Universal Robots PolyScope program: gravityFeederT.urp

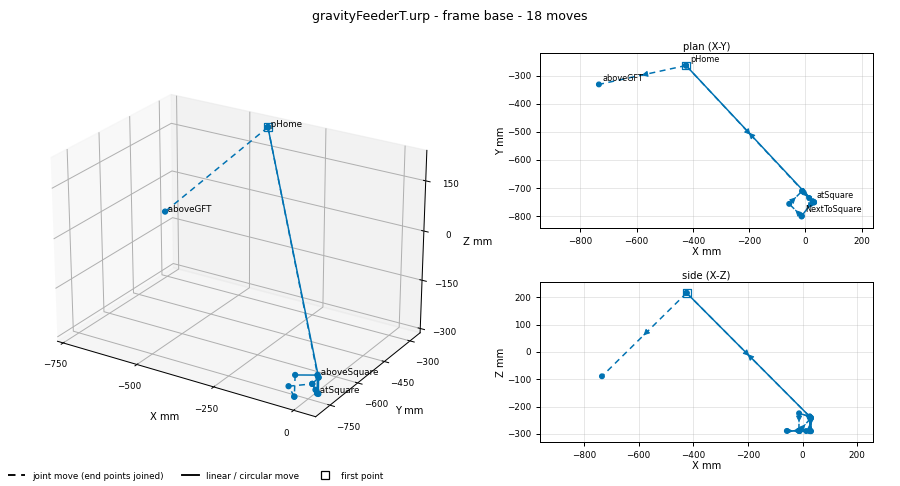
[picture p0: tool path of gravityFeederT.urp in frame base, 18 of 22 moves have a stored position in this frame; points joined in program order, loops and branches not executed]
Program gravityFeederT (installation=admin directory=/programs/THU_530PM createdIn=3.8.0.61336 lastSavedIn=3.15.8.106339 robotSerialNumber=2015350925)
Calibrated DH parameters: a=[0, -0.425, -0.39225, 0, 0, 0]; d=[0.089159, 0, 0, 0.10915, 0.09465, 0.0823]; alpha=[1.570796, 0, 0, 1.570796, -1.570796, 0]; deltaTheta=[0, 0, 0, 0, 0, 0]
Robot Program (runOnlyOnce=true)
  Set DigitalOutput pin=digital_out[0]; digitalValue=0
  Call _adminLinearIndex3
  MoveJ speed 180 deg/s, acceleration 100 deg/s^2 (useActiveTCP=true)
    Waypoint pHome: TCP in base x=-424.182 y=-264.292 z=215.908 mm, rx=-1.1973 ry=-2.8916 rz=-0.0083 rad; joints [224.997, -90.003, -90.003, -90.012, 89.253, -0.016] deg; flange x=-422.241 y=-266.331 z=431.79 mm, rx=-1.1973 ry=-2.8916 rz=-0.0083 rad
    Waypoint aboveGFT: TCP in base x=-733.795 y=-331.415 z=-88.949 mm, rx=-1.1406 ry=-2.7542 rz=0.4281 rad; joints [210.705, -134.689, -80.34, -37.4, 93.732, -13.725] deg; flange x=-685.048 y=-286.122 z=116.441 mm, rx=-1.1406 ry=-2.7542 rz=0.4281 rad
  MoveL speed 250 mm/s, acceleration 1200 mm/s^2 (useActiveTCP=true) feature=Base
    Waypoint atGFRel (Relative): relativeFromPosition TCP in base x=-734.776 y=-331.124 z=-89.043 mm, rx=-1.1456 ry=-2.7528 rz=0.4318 rad; joints [210.705, -134.689, -80.338, -37.4, 93.734, -13.726] deg; TCP in base x=-741.914 y=-341.01 z=-133.241 mm, rx=-1.1403 ry=-2.7544 rz=0.4285 rad; joints [211.023, -139.56, -78.724, -34.121, 93.656, -13.432] deg; flange x=-693.193 y=-295.644 z=72.139 mm, rx=-1.1403 ry=-2.7544 rz=0.4285 rad
    Set DigitalOutput pin=digital_out[0]; digitalValue=1
    Wait Sleep waitTime=1
    Waypoint moveUpRel (Relative): relativeFromPosition TCP in base x=-745.208 y=-342.748 z=-132.176 mm, rx=-1.1455 ry=-2.7527 rz=0.4317 rad; joints [211.078, -139.779, -78.056, -34.566, 93.626, -13.379] deg; TCP in base x=-747.389 y=-346.382 z=-130.447 mm, rx=-1.1404 ry=-2.7544 rz=0.4284 rad; joints [211.165, -140.11, -77.082, -35.205, 93.609, -13.293] deg; flange x=-698.665 y=-301.034 z=74.937 mm, rx=-1.1404 ry=-2.7544 rz=0.4284 rad
    Waypoint aboveGFRel (Relative): relativeFromPosition TCP in base x=-748.436 y=-346.052 z=-130.498 mm, rx=-1.1455 ry=-2.7528 rz=0.432 rad; joints [211.166, -140.109, -77.077, -35.205, 93.607, -13.294] deg; TCP in base x=-735.018 y=-332.975 z=-79.921 mm, rx=-1.1405 ry=-2.7541 rz=0.4282 rad; joints [210.763, -134.184, -79.714, -38.519, 93.714, -13.672] deg; flange x=-686.249 y=-287.668 z=125.46 mm, rx=-1.1405 ry=-2.7541 rz=0.4282 rad
  MoveJ speed 60 deg/s, acceleration 80 deg/s^2 (useActiveTCP=true)
    Waypoint pHome: TCP in base x=-424.182 y=-264.292 z=215.908 mm, rx=-1.1973 ry=-2.8916 rz=-0.0083 rad; joints [224.997, -90.003, -90.003, -90.012, 89.253, -0.016] deg; flange x=-422.241 y=-266.331 z=431.79 mm, rx=-1.1973 ry=-2.8916 rz=-0.0083 rad
    Waypoint aboveSquare: TCP in base x=26.216 y=-747.519 z=-236.314 mm, rx=1.1978 ry=2.9038 rz=-0.0039 rad; joints [280.423, -146.327, -75.803, -47.738, 89.943, 55.254] deg; flange x=26.339 y=-746.992 z=-20.414 mm, rx=1.1978 ry=2.9038 rz=-0.0039 rad
  MoveL speed 250 mm/s, acceleration 1200 mm/s^2 (useActiveTCP=true) feature=Base
    Waypoint atSquare: TCP in base x=26.393 y=-747.516 z=-289.105 mm, rx=1.1975 ry=2.9036 rz=-0.0037 rad; joints [280.428, -151.459, -74.791, -43.615, 89.962, 55.25] deg; flange x=26.44 y=-746.992 z=-73.206 mm, rx=1.1975 ry=2.9036 rz=-0.0037 rad
    Set DigitalOutput pin=digital_out[0]; digitalValue=0
    Wait Sleep waitTime=1
    Waypoint aboveSquare: TCP in base x=26.216 y=-747.519 z=-236.314 mm, rx=1.1978 ry=2.9038 rz=-0.0039 rad; joints [280.423, -146.327, -75.803, -47.738, 89.943, 55.254] deg; flange x=26.339 y=-746.992 z=-20.414 mm, rx=1.1978 ry=2.9038 rz=-0.0039 rad
    Waypoint NextToSquare: TCP in base x=-12.707 y=-798.202 z=-224.352 mm, rx=1.1986 ry=2.9037 rz=-0.0039 rad; joints [276.969, -151.006, -63.38, -55.484, 89.941, 51.827] deg; flange x=-12.546 y=-797.69 z=-8.453 mm, rx=1.1986 ry=2.9037 rz=-0.0039 rad
    Set DigitalOutput pin=digital_out[0]; digitalValue=1
  MoveJ speed 180 deg/s, acceleration 100 deg/s^2 (useActiveTCP=true)
    Waypoint besideSquareY: TCP in base x=-13.325 y=-800.324 z=-287.966 mm, rx=1.1979 ry=2.9037 rz=-0.0036 rad; joints [276.899, -157.027, -61.628, -51.215, 89.96, 51.735] deg; flange x=-13.233 y=-799.823 z=-72.067 mm, rx=1.1979 ry=2.9037 rz=-0.0036 rad
  Wait Sleep waitTime=0.1
  MoveL speed 30 mm/s, acceleration 30 mm/s^2 (useActiveTCP=true) feature=Base
    If force()≤45 (checkContinuously=true)
      Waypoint atSquareY (Relative): relativeFromPosition TCP in base x=-14.016 y=-801.018 z=-288.29 mm, rx=1.2024 ry=2.8992 rz=-0.0032 rad; joints [276.894, -157.026, -61.631, -51.22, 89.955, 51.756] deg; TCP in base x=0.346 y=-786.377 z=-288.706 mm, rx=1.1983 ry=2.9036 rz=-0.0038 rad; joints [278.023, -155.453, -65.375, -49.041, 89.95, 52.874] deg; flange x=0.463 y=-785.86 z=-72.807 mm, rx=1.1983 ry=2.9036 rz=-0.0038 rad
    Wait Sleep waitTime=0.5
  MoveJ speed 180 deg/s, acceleration 100 deg/s^2 (useActiveTCP=true)
    Waypoint besideSquareY: TCP in base x=-13.325 y=-800.324 z=-287.966 mm, rx=1.1979 ry=2.9037 rz=-0.0036 rad; joints [276.899, -157.027, -61.628, -51.215, 89.96, 51.735] deg; flange x=-13.233 y=-799.823 z=-72.067 mm, rx=1.1979 ry=2.9037 rz=-0.0036 rad
    Waypoint linkingMove: motionParameters(blendRadius=0.005); TCP in base x=-57.473 y=-755.963 z=-288.81 mm, rx=1.1976 ry=2.9038 rz=-0.0034 rad; joints [273.941, -152.445, -72.394, -45.037, 89.973, 48.766] deg; flange x=-57.402 y=-755.491 z=-72.91 mm, rx=1.1976 ry=2.9038 rz=-0.0034 rad
    Waypoint besideSquareX: TCP in base x=-11.173 y=-709.987 z=-289.359 mm, rx=1.1971 ry=2.9038 rz=-0.0033 rad; joints [277.951, -148.014, -83.176, -38.685, 89.975, 52.76] deg; flange x=-11.144 y=-709.507 z=-73.459 mm, rx=1.1971 ry=2.9038 rz=-0.0033 rad
  Wait Sleep waitTime=0.1
  MoveL speed 30 mm/s, acceleration 30 mm/s^2 (useActiveTCP=true) feature=Base
    If force()≤45 (checkContinuously=true)
      Waypoint atSquareX: TCP in base x=13.324 y=-734.787 z=-289.281 mm, rx=1.1981 ry=2.9035 rz=-0.0034 rad; joints [279.595, -150.232, -77.756, -41.889, 89.962, 54.442] deg; flange x=13.386 y=-734.31 z=-73.382 mm, rx=1.1981 ry=2.9035 rz=-0.0034 rad
    Wait Sleep waitTime=0.5
  MoveJ speed 60 deg/s, acceleration 80 deg/s^2 (useActiveTCP=true)
    Waypoint besideSquareX: TCP in base x=-11.173 y=-709.987 z=-289.359 mm, rx=1.1971 ry=2.9038 rz=-0.0033 rad; joints [277.951, -148.014, -83.176, -38.685, 89.975, 52.76] deg; flange x=-11.144 y=-709.507 z=-73.459 mm, rx=1.1971 ry=2.9038 rz=-0.0033 rad
    Waypoint aboveSquare2: TCP in base x=30.88 y=-750.293 z=-240.917 mm, rx=1.1981 ry=2.904 rz=-0.0037 rad; joints [280.742, -147.07, -75.056, -47.757, 89.931, 55.58] deg; flange x=31.053 y=-749.81 z=-25.017 mm, rx=1.1981 ry=2.904 rz=-0.0037 rad
    Set DigitalOutput pin=digital_out[0]; digitalValue=0
    Wait Sleep waitTime=1
  MoveL speed 250 mm/s, acceleration 1200 mm/s^2 (useActiveTCP=true) feature=Base
    Waypoint atSquare2: TCP in base x=31.052 y=-750.352 z=-289.802 mm, rx=1.1976 ry=2.904 rz=-0.0037 rad; joints [280.75, -151.826, -74.062, -43.986, 89.943, 55.574] deg; flange x=31.177 y=-749.848 z=-73.903 mm, rx=1.1976 ry=2.904 rz=-0.0037 rad
    Set DigitalOutput pin=digital_out[0]; digitalValue=1
    Wait Sleep waitTime=1
    Waypoint easeout: TCP in base x=27.298 y=-750.335 z=-289.811 mm, rx=1.1977 ry=2.904 rz=-0.0036 rad; joints [280.465, -151.813, -74.095, -43.971, 89.943, 55.29] deg; flange x=27.425 y=-749.847 z=-73.911 mm, rx=1.1977 ry=2.904 rz=-0.0036 rad
    Waypoint aboveSquare2: TCP in base x=30.88 y=-750.293 z=-240.917 mm, rx=1.1981 ry=2.904 rz=-0.0037 rad; joints [280.742, -147.07, -75.056, -47.757, 89.931, 55.58] deg; flange x=31.053 y=-749.81 z=-25.017 mm, rx=1.1981 ry=2.904 rz=-0.0037 rad
  MoveL speed 250 mm/s, acceleration 1200 mm/s^2 (useActiveTCP=true) feature=Base
    Waypoint pHome: TCP in base x=-424.182 y=-264.292 z=215.908 mm, rx=-1.1973 ry=-2.8916 rz=-0.0083 rad; joints [224.997, -90.003, -90.003, -90.012, 89.253, -0.016] deg; flange x=-422.241 y=-266.331 z=431.79 mm, rx=-1.1973 ry=-2.8916 rz=-0.0083 rad
SubProgram -> _adminLinearIndex3
SubProgram _adminLinearIndex3 (keepSynchronizedWithDisk=false) programFile=/programs/me345_admin/_adminLinearIndex3.urp
  Folder Move_linear_slide_Index3
    var_1 := False
    Loop While (checkContinuously=false) expression=var_1≟ False
      var_1 := socket_open("10.241.34.48",4001)
    var_3 := 1
    Send := "s r0x24 21"
    Script: socket_send_string(Send)
    Script: socket_send_byte(13)
    Send_Reply := socket_read_string()
    Send := "s r0xca 112778"
    Script: socket_send_string(Send)
    Script: socket_send_byte(13)
    Send_Reply := socket_read_string()
    Send := "t 1"
    Script: socket_send_string(Send)
    Script: socket_send_byte(13)
    Send_Reply := socket_read_string()
    Loop While (checkContinuously=false) expression=var_3≠0
      Send := "g r0xA0"
      Script: socket_send_string(Send)
      Script: socket_send_byte(13)
      var_3 := socket_get_var("v")
      Wait Sleep waitTime=0.1
    Script: socket_close()
    Script: sync()
